(* Logix 5000 project; controller CLP_AB vendor 1 type 14 code 79 rev 17.4; software revision 17.01 *)

TASK DeviceNet (continuous, watchdog 500 ms) : DeviceN
TASK Initialize_speed (event, rate 10 ms, priority 10, watchdog 500 ms) : Initialize_Data
TASK MainTask (periodic, rate 50 ms, priority 10, watchdog 500 ms) : Camera_Trigger

MODULES
   Local : vendor 1 type 14 code 79 (ICP 0, rev 17.4)
      DN : vendor 1 type 12 code 14 (ICP 2, rev 7.3, Output RPI 20 ms, Input RPI 20 ms)
      Ethernet : 1756-ENBT (Ethernet 192.168.0.4, ICP 3, rev 4.1)
         Camera_Sensor : ETHERNET-MODULE (Ethernet 192.168.0.3, rev 1.1, Output RPI 25 ms)   // Banner
      LocalSERCOS : vendor 1 type 16 code 14 (ICP 1, rev 17.2, MotionAsync RPI 25 ms, MotionEvent RPI 1000 ms, MotionSync RPI 2 ms)
         Drive : vendor 1 type 115 code 164 (SERCOS 1, rev 1.1)
END_MODULES

VAR_GLOBAL   (* controller tags *)
   BitTest1 : BOOL;
   BitTest2 : BOOL;
   botao : BOOL;
   currentSpeedTopo : REAL;
   dataInitialized : BOOL;
   dir_int : DINT;
   direction : BOOL;
   drive_axis : AXIS_SERVO_DRIVE;
   dt : REAL;
   Emanuel : BOOL;
   encoder : AXIS_SERVO_DRIVE;
   IterationChange : ALIAS FOR Camera_Sensor:I.Data[6].0;
   IterationChanged : BOOL;
   IterationCount : DINT;
   lastIterationCount : DINT;
   MAH_0 : MOTION_INSTRUCTION;
   MAJ_0 : MOTION_INSTRUCTION := (FLAGS := 33554432);
   MAJ_1 : MOTION_INSTRUCTION := (FLAGS := 33554432);
   MAJ_2 : MOTION_INSTRUCTION;
   MAS_0 : MOTION_INSTRUCTION;
   MAS_1 : MOTION_INSTRUCTION := (FLAGS := 33554432);
   MAS_2 : MOTION_INSTRUCTION;
   MGroup : MOTION_GROUP;
   MSF_0 : MOTION_INSTRUCTION;
   MSO_0 : MOTION_INSTRUCTION;
   MSO_1 : MOTION_INSTRUCTION := (FLAGS := -1610612736, EN := 1, DN := 1, STATE := 1);
   OutTest1 : BOOL;
   OutTest2 : BOOL;
   position_fundo : REAL[342];
   position_topo : REAL[342];
   positionFundo : ALIAS FOR Camera_Sensor:I.Data[16];
   pyTrigger : BOOL;
   Ready : ALIAS FOR Camera_Sensor:I.Data[0].4;
   refPositionFundo : REAL;
   speed : REAL[342];
   speedRate : REAL;
   timer_1 : TIMER := (PRE := 500);
   Trigger_ACK : ALIAS FOR Camera_Sensor:I.Data[0].16;
   trigger_off : TIMER := (PRE := 10);
   trigger_on : TIMER := (PRE := 10);
END_VAR

PROGRAM Camera_Trigger   (* main routine TriggerMain *)
// Trigger
VAR
   Trigger : ALIAS FOR Camera_Sensor:O.Data[0].0;
END_VAR

ROUTINE TriggerMain   (* ladder *)
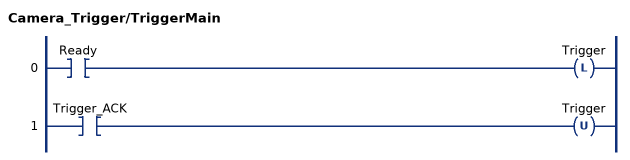
   0: XIC(Ready)OTL(Trigger);
   1: XIC(Trigger_ACK)OTU(Trigger);
END_ROUTINE
END_PROGRAM

PROGRAM Controle   (* main routine malhaAberta *)
VAR
   direcMove : DINT;
   k : DINT;
   timervel : FBD_TIMER;
END_VAR

ROUTINE ControleMain   (* structured text *)
   COP(Camera_Sensor:I.Data[6],IterationCount,32);
   if IterationCount > lastIterationCount then
   	/*Aqui vai o nosso controlador*/
   	if positionFundo > 205.0 then
   		speedRate:=.2;
   		direcMove:=1;
   	elsif positionFundo < 195.0 then
   		speedRate:=.2;
   		direcMove:=0;
   	else
   		speedRate:=0;
   		MAS(drive_axis,MAS_1,0,0,100,1,0,100,1);
   	end_if;
   	MAJ(drive_axis,MAJ_1,direcMove,speedRate,0,50.0,1,50.0,1,0,50.0,50.0,1,0,0);
   	COP(Camera_Sensor:I.Data[6],lastIterationCount,32);
   end_if;
END_ROUTINE

ROUTINE malhaAberta   (* structured text *)
   // k is the index of the speed vector
   if dataInitialized AND k < 140 then
   	currentSpeedTopo := speed[k];
   	refPositionFundo := position_fundo[k];
   	MAJ(drive_axis,MAJ_1,0,speed[k],0,50.0,1,50.0,1,0,50.0,50.0,1,0,0);
   	k:=k + 1;
   end_if;
   
   if k >= 85 then
   	MAS(drive_axis,MAS_1,0,0,100,1,0,100,1);
   	if MAS_1.DN then
   		MSF(drive_axis,MSF_0);
   	end_if;
   end_if;
END_ROUTINE

ROUTINE VeloMain   (* structured text *)
   COP(Camera_Sensor:I.Data[6],IterationCount,32);
   /*MAJ(drive_axis,MAJ_1,0,0.5,0,50.0,1,50.0,1,0,50.0,50.0,1,0,0);
   timervel.TimerEnable:=1;
   TONR(timervel);
   MAS(drive_axis,MAS_1,All,0,100,1,0,100,1);
   MSF(drive_axis,MSF_0);
   */
   	//MSO(drive_axis,MSO_1);
   	timervel.PRE:=20000;
   	if (MSO_1.EN AND timervel.ACC < 20000) then
   		if (NOT timervel.DN) then
   			timervel.TimerEnable:=1;
   			MAJ(drive_axis,MAJ_1,0,0.2,0,50.0,1,50.0,1,0,50.0,50.0,1,0,0);
   			TONR(timervel);
   		end_if;
   	end_if;
   	if (timervel.DN) then
   		MAS(drive_axis,MAS_1,All,0,100,1,0,100,1);
   	end_if;
   	if (MAS_1.EN) then
   		MSF(drive_axis,MSF_0);
   	end_if;
   
END_ROUTINE
END_PROGRAM

PROGRAM Controle1   (* main routine VeloMain *)
VAR
   direcMove : DINT;
   timervel : FBD_TIMER;
END_VAR

ROUTINE ControleMain   (* structured text *)
   COP(Camera_Sensor:I.Data[6],IterationCount,32);
   if IterationCount > lastIterationCount then
   	/*Aqui vai o nosso controlador*/
   	if positionFundo > 205.0 then
   		speedRate:=.2;
   		direcMove:=1;
   	elsif positionFundo < 195.0 then
   		speedRate:=.2;
   		direcMove:=0;
   	else
   		speedRate:=0;
   		MAS(drive_axis,MAS_1,0,0,100,1,0,100,1);
   	end_if;
   	MAJ(drive_axis,MAJ_1,direcMove,speedRate,0,50.0,1,50.0,1,0,50.0,50.0,1,0,0);
   	COP(Camera_Sensor:I.Data[6],lastIterationCount,32);
   end_if;
END_ROUTINE

ROUTINE VeloMain   (* structured text *)
   COP(Camera_Sensor:I.Data[6],IterationCount,32);
   /*MAJ(drive_axis,MAJ_1,0,0.5,0,50.0,1,50.0,1,0,50.0,50.0,1,0,0);
   timervel.TimerEnable:=1;
   TONR(timervel);
   MAS(drive_axis,MAS_1,All,0,100,1,0,100,1);
   MSF(drive_axis,MSF_0);
   */
   	//MSO(drive_axis,MSO_1);
   	timervel.PRE:=20000;
   	if (MSO_1.EN AND timervel.ACC < 20000) then
   		if (NOT timervel.DN) then
   			timervel.TimerEnable:=1;
   			MAJ(drive_axis,MAJ_1,0,0.2,0,50.0,1,50.0,1,0,50.0,50.0,1,0,0);
   			TONR(timervel);
   		end_if;
   	end_if;
   	if (timervel.DN) then
   		MAS(drive_axis,MAS_1,All,0,100,1,0,100,1);
   	end_if;
   	if (MAS_1.EN) then
   		MSF(drive_axis,MSF_0);
   	end_if;
   
END_ROUTINE
END_PROGRAM

PROGRAM DeviceN   (* main routine InitDNetST *)

ROUTINE InitDNetST   (* structured text *)
   Local:2:O.CommandRegister.Run [:=] 1;
   if (pyTrigger) AND (NOT dataInitialized) then
   	EVENT(Initialize_speed);
   end_if;
   
END_ROUTINE
END_PROGRAM

PROGRAM Initialize_Data   (* main routine Init *)

ROUTINE Init   (* structured text *)
   /* Universidade de Brasilia
   Trabalho de Graduacao em Engenharia Mecatronica
   Alunos:
   Ataias Pereira Reis 10/0093817
   Emanuel Pereira Barroso Neto 11/0115716
   This code must be executed only once. */
   
   MSO(drive_axis,MSO_1);
   
   /*Passo de tempo em segundos*/
   dt := 0.05;
   
   /*Velocidade esta em unidades/s*/
   speed[0] := 0.0;
   speed[1] := 0.0;
   speed[2] := 0.0;
   speed[3] := 0.0;
   speed[4] := 0.0;
   speed[5] := 0.0;
   speed[6] := 0.0;
   speed[7] := 0.0;
   speed[8] := 0.0;
   speed[9] := 0.0;
   speed[10] := 0.0;
   speed[11] := 0.0;
   speed[12] := 0.0;
   speed[13] := 0.0;
   speed[14] := 0.0;
   speed[15] := 0.0;
   speed[16] := 0.0;
   speed[17] := 0.0;
   speed[18] := 0.0517676857626;
   speed[19] := 0.124879505781;
   speed[20] := 0.207600335504;
   speed[21] := 0.295968298113;
   speed[22] := 0.389241858771;
   speed[23] := 0.48656581719;
   speed[24] := 0.587084307886;
   speed[25] := 0.689935515172;
   speed[26] := 0.794252492077;
   speed[27] := 0.899166493361;
   speed[28] := 1.00383634774;
   speed[29] := 1.10744817531;
   speed[30] := 1.20953872081;
   speed[31] := 1.30556546851;
   speed[32] := 1.38176888339;
   speed[33] := 1.44412814736;
   speed[34] := 1.51340846996;
   speed[35] := 1.5929293696;
   speed[36] := 1.6792516782;
   speed[37] := 1.76914619866;
   speed[38] := 1.85962724351;
   speed[39] := 1.94803310979;
   speed[40] := 2.03210211549;
   speed[41] := 2.10997477267;
   speed[42] := 2.18042256805;
   speed[43] := 2.2418987926;
   speed[44] := 2.29552201078;
   speed[45] := 2.33907631965;
   speed[46] := 2.36759784772;
   speed[47] := 2.38339114539;
   speed[48] := 2.38649362399;
   speed[49] := 2.37754921271;
   speed[50] := 2.35722506482;
   speed[51] := 2.32540404626;
   speed[52] := 2.28281415338;
   speed[53] := 2.23104367474;
   speed[54] := 2.1704473561;
   speed[55] := 2.10187462449;
   speed[56] := 2.02690935379;
   speed[57] := 1.94551390162;
   speed[58] := 1.85867695573;
   speed[59] := 1.76772327269;
   speed[60] := 1.67552357606;
   speed[61] := 1.58086227538;
   speed[62] := 1.48437915097;
   speed[63] := 1.38868886367;
   speed[64] := 1.29243567476;
   speed[65] := 1.19761963512;
   speed[66] := 1.10732868951;
   speed[67] := 1.01873221001;
   speed[68] := 0.9319276396;
   speed[69] := 0.847517232811;
   speed[70] := 0.767251289573;
   speed[71] := 0.694157750934;
   speed[72] := 0.621707544577;
   speed[73] := 0.548114277662;
   speed[74] := 0.482264121959;
   speed[75] := 0.417503469359;
   speed[76] := 0.355331643999;
   speed[77] := 0.297736171581;
   speed[78] := 0.245060897905;
   speed[79] := 0.198152036973;
   speed[80] := 0.155377487622;
   speed[81] := 0.122729213657;
   speed[82] := 0.0881979949101;
   speed[83] := 0.0595774855511;
   speed[84] := 0.0;
   speed[85] := 0.0;
   speed[86] := 0.0;
   speed[87] := 0.0;
   speed[88] := 0.0;
   speed[89] := 0.0;
   speed[90] := 0.0;
   speed[91] := 0.0;
   speed[92] := 0.0;
   speed[93] := 0.0;
   speed[94] := 0.0;
   speed[95] := 0.0;
   speed[96] := 0.0;
   speed[97] := 0.0;
   speed[98] := 0.0;
   speed[99] := 0.0;
   speed[100] := 0.0;
   speed[101] := 0.0;
   speed[102] := 0.0;
   speed[103] := 0.0;
   speed[104] := 0.0;
   speed[105] := 0.0;
   speed[106] := 0.0;
   speed[107] := 0.0;
   speed[108] := 0.0;
   speed[109] := 0.0;
   speed[110] := 0.0;
   speed[111] := 0.0;
   speed[112] := 0.0;
   speed[113] := 0.0;
   speed[114] := 0.0;
   speed[115] := 0.0;
   speed[116] := 0.0;
   speed[117] := 0.0;
   speed[118] := 0.0;
   speed[119] := 0.0;
   speed[120] := 0.0;
   speed[121] := 0.0;
   speed[122] := 0.0;
   speed[123] := 0.0;
   speed[124] := 0.0;
   speed[125] := 0.0;
   speed[126] := 0.0;
   speed[127] := 0.0;
   speed[128] := 0.0;
   speed[129] := 0.0;
   speed[130] := 0.0;
   speed[131] := 0.0;
   speed[132] := 0.0;
   speed[133] := 0.0;
   speed[134] := 0.0;
   speed[135] := 0.0;
   speed[136] := 0.0;
   speed[137] := 0.0;
   speed[138] := 0.0;
   speed[139] := 0.0;
   
   /*Posicao esta em mm*/
   position_topo[0] := 0.0;
   position_topo[1] := 0.0;
   position_topo[2] := 0.0;
   position_topo[3] := 0.0;
   position_topo[4] := 0.0;
   position_topo[5] := 0.0;
   position_topo[6] := 0.0;
   position_topo[7] := 0.0;
   position_topo[8] := 0.0;
   position_topo[9] := 0.0;
   position_topo[10] := 0.0;
   position_topo[11] := 0.0;
   position_topo[12] := 0.0;
   position_topo[13] := 0.0;
   position_topo[14] := 0.0;
   position_topo[15] := 0.0;
   position_topo[16] := 0.0;
   position_topo[17] := 0.0;
   position_topo[18] := 0.0;
   position_topo[19] := 0.0;
   position_topo[20] := 0.00100277197087;
   position_topo[21] := 0.00189907823213;
   position_topo[22] := 0.00311949109903;
   position_topo[23] := 0.00467999630258;
   position_topo[24] := 0.00659351710071;
   position_topo[25] := 0.00886990646408;
   position_topo[26] := 0.0115159378109;
   position_topo[27] := 0.0145352895283;
   position_topo[28] := 0.017928575326;
   position_topo[29] := 0.0216934873631;
   position_topo[30] := 0.0258247579254;
   position_topo[31] := 0.0303126352038;
   position_topo[32] := 0.0351133538009;
   position_topo[33] := 0.0401515025198;
   position_topo[34] := 0.0454206619227;
   position_topo[35] := 0.0509568206355;
   position_topo[36] := 0.0567896198594;
   position_topo[37] := 0.0629376256869;
   position_topo[38] := 0.0694080497261;
   position_topo[39] := 0.0761982019533;
   position_topo[40] := 0.0832964669918;
   position_topo[41] := 0.0906839706072;
   position_topo[42] := 0.0983362113297;
   position_topo[43] := 0.10622435959;
   position_topo[44] := 0.114315947463;
   position_topo[45] := 0.122584410213;
   position_topo[46] := 0.13098050947;
   position_topo[47] := 0.139455336989;
   position_topo[48] := 0.147963967058;
   position_topo[49] := 0.156461659758;
   position_topo[50] := 0.164907330411;
   position_topo[51] := 0.173259931818;
   position_topo[52] := 0.181479523576;
   position_topo[53] := 0.189530177893;
   position_topo[54] := 0.197381086792;
   position_topo[55] := 0.205000470545;
   position_topo[56] := 0.212364253427;
   position_topo[57] := 0.219448899232;
   position_topo[58] := 0.226233452467;
   position_topo[59] := 0.232700218137;
   position_topo[60] := 0.238839515145;
   position_topo[61] := 0.244647233479;
   position_topo[62] := 0.250112311987;
   position_topo[63] := 0.255234721393;
   position_topo[64] := 0.260015995116;
   position_topo[65] := 0.264454114813;
   position_topo[66] := 0.268562829301;
   position_topo[67] := 0.27235364047;
   position_topo[68] := 0.275830814572;
   position_topo[69] := 0.279003137764;
   position_topo[70] := 0.281880108649;
   position_topo[71] := 0.284483487184;
   position_topo[72] := 0.286831917376;
   position_topo[73] := 0.288916351638;
   position_topo[74] := 0.290750556885;
   position_topo[75] := 0.292356736364;
   position_topo[76] := 0.293731989009;
   position_topo[77] := 0.294896004348;
   position_topo[78] := 0.295861280634;
   position_topo[79] := 0.296651219901;
   position_topo[80] := 0.297278491208;
   position_topo[81] := 0.297771971864;
   position_topo[82] := 0.29815131277;
   position_topo[83] := 0.298408218512;
   position_topo[84] := 0.298592150875;
   position_topo[85] := 0.298725420273;
   position_topo[86] := 0.298797884919;
   position_topo[87] := 0.298817025596;
   position_topo[88] := 0.298799262345;
   position_topo[89] := 0.298789121463;
   position_topo[90] := 0.298799608473;
   position_topo[91] := 0.298813457704;
   position_topo[92] := 0.298829892846;
   position_topo[93] := 0.298840159831;
   position_topo[94] := 0.298834543546;
   position_topo[95] := 0.298829977228;
   position_topo[96] := 0.298863174567;
   position_topo[97] := 0.298929605231;
   position_topo[98] := 0.298997700728;
   position_topo[99] := 0.299031337491;
   position_topo[100] := 0.299011937976;
   position_topo[101] := 0.298989284721;
   position_topo[102] := 0.299045197966;
   position_topo[103] := 0.299092747998;
   position_topo[104] := 0.299068748259;
   position_topo[105] := 0.2990784776;
   position_topo[106] := 0.299124926652;
   position_topo[107] := 0.299085722425;
   position_topo[108] := 0.299099905779;
   position_topo[109] := 0.29912782583;
   position_topo[110] := 0.299108597793;
   position_topo[111] := 0.299165572936;
   position_topo[112] := 0.299113585782;
   position_topo[113] := 0.299123304013;
   position_topo[114] := 0.299146010228;
   position_topo[115] := 0.299176817206;
   position_topo[116] := 0.29917810103;
   position_topo[117] := 0.299193651839;
   position_topo[118] := 0.299225472016;
   position_topo[119] := 0.299253479086;
   position_topo[120] := 0.299259821075;
   position_topo[121] := 0.29927998091;
   position_topo[122] := 0.299296273361;
   position_topo[123] := 0.299318577393;
   position_topo[124] := 0.299279940553;
   position_topo[125] := 0.299253209986;
   position_topo[126] := 0.299200164256;
   position_topo[127] := 0.299220513468;
   position_topo[128] := 0.299275386106;
   position_topo[129] := 0.299267030823;
   position_topo[130] := 0.299238268735;
   position_topo[131] := 0.299264131385;
   position_topo[132] := 0.299278973465;
   position_topo[133] := 0.299244209158;
   position_topo[134] := 0.299287092298;
   position_topo[135] := 0.299306272694;
   position_topo[136] := 0.299292804028;
   position_topo[137] := 0.299336184009;
   position_topo[138] := 0.299307968378;
   position_topo[139] := 0.299349900916;
   
   position_fundo[0] := 0.0;
   position_fundo[1] := 0.0;
   position_fundo[2] := 0.0;
   position_fundo[3] := 0.0;
   position_fundo[4] := 0.0;
   position_fundo[5] := 0.0;
   position_fundo[6] := 0.0;
   position_fundo[7] := 0.0;
   position_fundo[8] := 0.0;
   position_fundo[9] := 0.0;
   position_fundo[10] := 0.0;
   position_fundo[11] := 0.0;
   position_fundo[12] := 0.0;
   position_fundo[13] := 0.0;
   position_fundo[14] := 0.0;
   position_fundo[15] := 0.0;
   position_fundo[16] := 0.0;
   position_fundo[17] := 0.0;
   position_fundo[18] := 0.0;
   position_fundo[19] := 0.0;
   position_fundo[20] := 0.0;
   position_fundo[21] := 0.0;
   position_fundo[22] := 0.0;
   position_fundo[23] := 0.0;
   position_fundo[24] := 0.0;
   position_fundo[25] := 0.0;
   position_fundo[26] := 0.0;
   position_fundo[27] := 0.0;
   position_fundo[28] := 0.0;
   position_fundo[29] := 0.00153550911288;
   position_fundo[30] := 0.0029627797267;
   position_fundo[31] := 0.00500541576333;
   position_fundo[32] := 0.0077237286035;
   position_fundo[33] := 0.0111588517211;
   position_fundo[34] := 0.0153344488369;
   position_fundo[35] := 0.0202584470826;
   position_fundo[36] := 0.0259246651982;
   position_fundo[37] := 0.0323143659097;
   position_fundo[38] := 0.0393977294747;
   position_fundo[39] := 0.0471352942596;
   position_fundo[40] := 0.0554793501137;
   position_fundo[41] := 0.0643752433166;
   position_fundo[42] := 0.0737626162585;
   position_fundo[43] := 0.0835765832539;
   position_fundo[44] := 0.0937488654491;
   position_fundo[45] := 0.104208850553;
   position_fundo[46] := 0.114884585156;
   position_fundo[47] := 0.125703707206;
   position_fundo[48] := 0.136594321755;
   position_fundo[49] := 0.147485809035;
   position_fundo[50] := 0.158309567294;
   position_fundo[51] := 0.168999695134;
   position_fundo[52] := 0.179493622306;
   position_fundo[53] := 0.189732665002;
   position_fundo[54] := 0.199662515149;
   position_fundo[55] := 0.209233671782;
   position_fundo[56] := 0.218401818455;
   position_fundo[57] := 0.227128141219;
   position_fundo[58] := 0.235379560061;
   position_fundo[59] := 0.243128908735;
   position_fundo[60] := 0.25035505605;
   position_fundo[61] := 0.257042978906;
   position_fundo[62] := 0.263183751893;
   position_fundo[63] := 0.268774468825;
   position_fundo[64] := 0.273818112944;
   position_fundo[65] := 0.278323370746;
   position_fundo[66] := 0.282304387532;
   position_fundo[67] := 0.285780434838;
   position_fundo[68] := 0.288775527888;
   position_fundo[69] := 0.291317984965;
   position_fundo[70] := 0.293439930471;
   position_fundo[71] := 0.295176723375;
   position_fundo[72] := 0.296566319466;
   position_fundo[73] := 0.297648580492;
   position_fundo[74] := 0.298464521481;
   position_fundo[75] := 0.299055490986;
   position_fundo[76] := 0.299462286308;
   position_fundo[77] := 0.299724212532;
   position_fundo[78] := 0.29987808035;
   position_fundo[79] := 0.299957131325;
   position_fundo[80] := 0.299989898966;
   position_fundo[81] := 0.299999020311;
   position_fundo[82] := 0.300000000026;
   position_fundo[83] := 0.300000000876;
   position_fundo[84] := 0.29999999969;
   position_fundo[85] := 0.300000000063;
   position_fundo[86] := 0.299999999993;
   position_fundo[87] := 0.3;
   position_fundo[88] := 0.3;
   position_fundo[89] := 0.3;
   position_fundo[90] := 0.3;
   position_fundo[91] := 0.3;
   position_fundo[92] := 0.3;
   position_fundo[93] := 0.3;
   position_fundo[94] := 0.3;
   position_fundo[95] := 0.3;
   position_fundo[96] := 0.3;
   position_fundo[97] := 0.3;
   position_fundo[98] := 0.3;
   position_fundo[99] := 0.3;
   position_fundo[100] := 0.3;
   position_fundo[101] := 0.3;
   position_fundo[102] := 0.3;
   position_fundo[103] := 0.3;
   position_fundo[104] := 0.3;
   position_fundo[105] := 0.3;
   position_fundo[106] := 0.3;
   position_fundo[107] := 0.3;
   position_fundo[108] := 0.3;
   position_fundo[109] := 0.3;
   position_fundo[110] := 0.3;
   position_fundo[111] := 0.3;
   position_fundo[112] := 0.3;
   position_fundo[113] := 0.3;
   position_fundo[114] := 0.3;
   position_fundo[115] := 0.3;
   position_fundo[116] := 0.3;
   position_fundo[117] := 0.3;
   position_fundo[118] := 0.3;
   position_fundo[119] := 0.3;
   position_fundo[120] := 0.3;
   position_fundo[121] := 0.3;
   position_fundo[122] := 0.3;
   position_fundo[123] := 0.3;
   position_fundo[124] := 0.3;
   position_fundo[125] := 0.3;
   position_fundo[126] := 0.3;
   position_fundo[127] := 0.3;
   position_fundo[128] := 0.3;
   position_fundo[129] := 0.3;
   position_fundo[130] := 0.3;
   position_fundo[131] := 0.3;
   position_fundo[132] := 0.3;
   position_fundo[133] := 0.3;
   position_fundo[134] := 0.3;
   position_fundo[135] := 0.3;
   position_fundo[136] := 0.3;
   position_fundo[137] := 0.3;
   position_fundo[138] := 0.3;
   position_fundo[139] := 0.3;
   
   
   dataInitialized := 1;
   
END_ROUTINE
END_PROGRAM

PROGRAM MainProgram   (* main routine MainRoutineST *)

ROUTINE MainRoutine   (* ladder *)
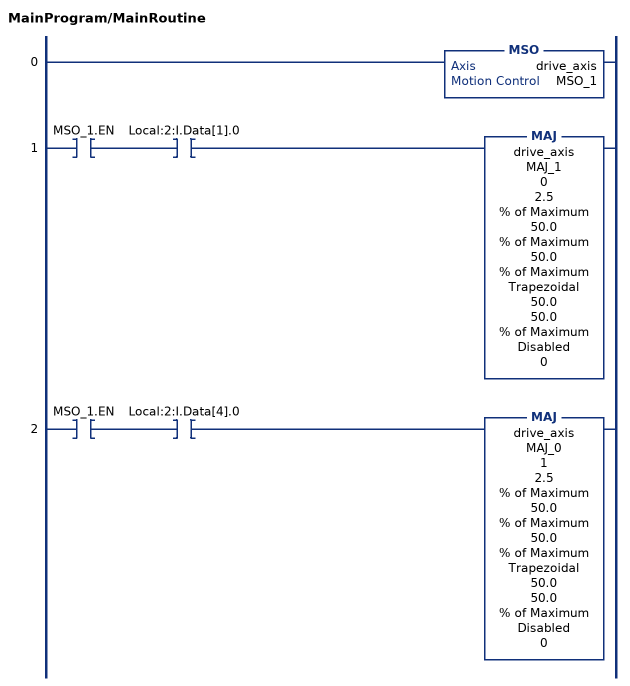
   0: MSO(drive_axis,MSO_1);
   1: XIC(MSO_1.EN)XIC(Local:2:I.Data[1].0)MAJ(drive_axis,MAJ_1,0,2.5,% of Maximum,50.0,% of Maximum,50.0,% of Maximum,Trapezoidal,50.0,50.0,% of Maximum,Disabled,0);
   2: XIC(MSO_1.EN)XIC(Local:2:I.Data[4].0)MAJ(drive_axis,MAJ_0,1,2.5,% of Maximum,50.0,% of Maximum,50.0,% of Maximum,Trapezoidal,50.0,50.0,% of Maximum,Disabled,0);
END_ROUTINE

ROUTINE MainRoutineST   (* structured text *)
   MSO(drive_axis,MSO_1);
   IF MSO_1.EN AND Local:2:I.Data[1].0 THEN
   	MAJ(drive_axis,MAJ_1,0,2.5,1,50.0,1,50.0,1,0,50.0,50.0,1,0,0);
   END_IF;
   IF MSO_1.EN AND Local:2:I.Data[4].0 THEN
   	MAJ(drive_axis,MAJ_0,1,2.5,1,50.0,1,50.0,1,0,50.0,50.0,1,0,0);
   END_IF;
END_ROUTINE
END_PROGRAM

PROGRAM Parada   (* main routine parada *)

ROUTINE parada   (* ladder *)
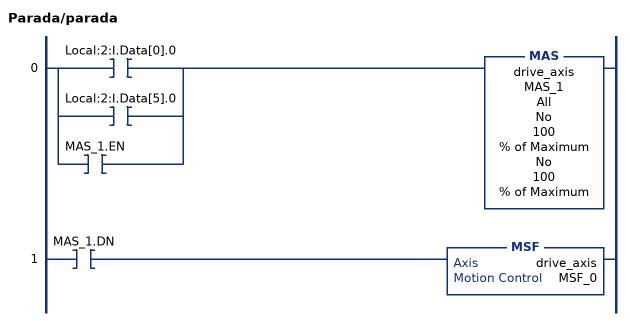
   0: [XIC(Local:2:I.Data[0].0) ,[XIC(Local:2:I.Data[5].0) ,XIC(MAS_1.EN) ] ]MAS(drive_axis,MAS_1,All,No,100,% of Maximum,No,100,% of Maximum);
   1: XIC(MAS_1.DN)MSF(drive_axis,MSF_0);
END_ROUTINE
END_PROGRAM
